# EPICS substitutions: DAS240/DAS240-IOC-01App/Db/DAS240A.substitutions
global{P=\$(P),C=\$(C),PORT=\$(PORT)}

file "Analogue.template" {
    pattern{ N, OFFSET }
    { 1, 0 }
    { 2, 2 }
    { 3, 4 }
    { 4, 6 }
    { 5, 8 }
    { 6, 10 }
    { 7, 12 }
    { 8, 14 }
    { 9, 16 }
    { 10, 18 }
    { 11, 20 }
    { 12, 22 }
    { 13, 24 }
    { 14, 26 }
    { 15, 28 }
    { 16, 30 }
    { 17, 32 }
    { 18, 34 }
    { 19, 36 }
    { 20, 38 }
}
